GLOBALCONSTANTS AID_NV (* Number variable object attribute ids (all read-only) *)
  (* Standard: 61499-1; Description: Copyright (c) 2023 HR Agrartechnik GmbH This program and the accompanying materials are made available under the terms of the Eclipse Public License 2.0 which is available at https://www.eclipse.org/legal/epl-2.0/ SPDX-License-Identifier: EPL-2.0 *)
  (* Version 1.0, 2026-06-20, Franz Höpfinger, HR Agrartechnik GmbH *)
  PACKAGE isobus::UT::Q::const::AID;
  VAR_GLOBAL CONSTANT
    VALUE : USINT := USINT#1; (* 1: AID_NV_VALUE (read-only) - Current value. *)
  END_VAR
END_GLOBALCONSTANTS
